KUKA KRL program: chk_w3_grp2_clo.src

&ACCESS RVO1
&COMMENT Check GRP Z2 ACTROS CLOSE
DEF chk_w3_grp2_clo( )

; Check gripper actros CLOSE Z2
;//---- Start User-------

$TIMER[10] = 0
$TIMER_STOP[10] = FALSE

WAIT FOR ($IN[10])
WAIT FOR (NOT $IN[9])

$TIMER_STOP[10] = TRUE
$TIMER[10] = 0

;//---- End User---------

END
